(* CoDeSys 2.3.9.62 project: DosVagones.pro *)
(* Libraries: Standard.lib 2.6.14 10:37:46, IecSfc.lib 2.6.14 11:37:46 *)

(* Global variable list: Global_Variables *)
VAR_GLOBAL

      (*Entradas*)
      P1:BOOL;
      P2:BOOL;
	A1:BOOL;
	B1:BOOL;
	A2:BOOL;
	B2:BOOL;

       (* Salidas *)
	MOTOR_IZ1:BOOL;
	MOTOR_DE1:BOOL;
       MOTOR_IZ2:BOOL;
	MOTOR_DE2:BOOL;
      Carga1:BOOL;
      Carga2:BOOL;
      Descarga1:BOOL;
      Descarga2:BOOL;

      (* Variables del simulador *)
	Vel:INT:=1;
	Vel2:INT:=1;
END_VAR

(* POU PLC_PRG, ST *)
PROGRAM PLC_PRG
VAR
END_VAR
Vehiculo();
Vehiculo2();

Automatismo;
END_PROGRAM

(* POU Vehiculo, ST *)
PROGRAM Vehiculo
VAR
	PosX: INT;
END_VAR
A1:=FALSE;
B1:=FALSE;


IF MOTOR_DE1=TRUE THEN

     PosX:=PosX+Vel;

END_IF

IF MOTOR_IZ1=TRUE THEN

     PosX:=PosX-Vel;

END_IF


IF PosX<=0 THEN
   A1:=TRUE;
END_IF

IF PosX>=400 THEN
  B1:=TRUE;
END_IF
END_PROGRAM

(* POU Vehiculo2, ST *)
PROGRAM Vehiculo2
VAR
	PosX2: INT;
END_VAR
A2:=FALSE;
B2:=FALSE;


IF MOTOR_DE2=TRUE THEN

     PosX2:=PosX2+Vel2;

END_IF

IF MOTOR_IZ2=TRUE THEN

     PosX2:=PosX2-Vel2;

END_IF


IF PosX2<=0 THEN
   A2:=TRUE;
END_IF

IF PosX2>=400 THEN
  B2:=TRUE;
END_IF
END_PROGRAM

(* POU Automatismo, LD *)
PROGRAM Automatismo
VAR
	Control1: controlVehiculo;
	Control2: ControlVehiculo;
	IniciaDescarga: BOOL;
	EnB2: BOOL;
	EnB1: BOOL;
END_VAR
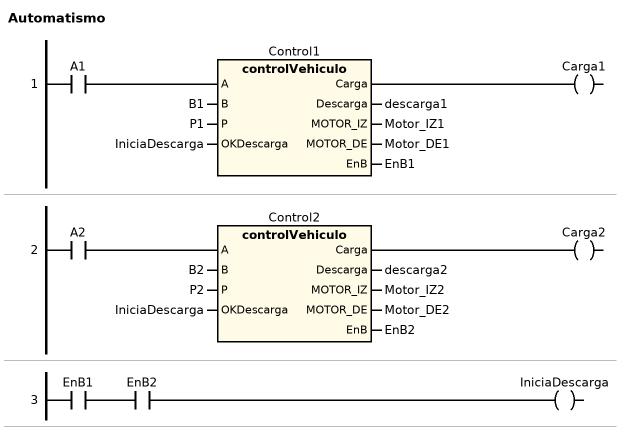
_LD_ (* Ladder Diagram *)
NETWORK 1
	[A1] - Control1:controlVehiculo(A: *, B: B1, P: P1, OKDescarga: IniciaDescarga, Descarga => descarga1, MOTOR_IZ => Motor_IZ1, MOTOR_DE => Motor_DE1, EnB => EnB1) --- (Carga1)
NETWORK 2
	[A2] - Control2:controlVehiculo(A: *, B: B2, P: P2, OKDescarga: IniciaDescarga, Descarga => descarga2, MOTOR_IZ => Motor_IZ2, MOTOR_DE => Motor_DE2, EnB => EnB2) --- (Carga2)
NETWORK 3
	[EnB1] - [EnB2] --- (IniciaDescarga)
_END_LD_
(* the same logic as Structured Text *)
(* Network 1 *)
Control1(A := A1, B := B1, P := P1, OKDescarga := IniciaDescarga);
descarga1 := Control1.Descarga;
Motor_IZ1 := Control1.MOTOR_IZ;
Motor_DE1 := Control1.MOTOR_DE;
EnB1 := Control1.EnB;
Carga1 := Control1.Carga;
(* Network 2 *)
Control2(A := A2, B := B2, P := P2, OKDescarga := IniciaDescarga);
descarga2 := Control2.Descarga;
Motor_IZ2 := Control2.MOTOR_IZ;
Motor_DE2 := Control2.MOTOR_DE;
EnB2 := Control2.EnB;
Carga2 := Control2.Carga;
(* Network 3 *)
IniciaDescarga := EnB1 AND EnB2;
END_PROGRAM

(* POU ControlVehiculo, LD *)
FUNCTION_BLOCK ControlVehiculo
VAR_INPUT
	A: BOOL;
	B: BOOL;
	P: BOOL;
	OKDescarga: BOOL;
END_VAR
VAR_OUTPUT
	Carga: BOOL;
	Descarga: BOOL;
	MOTOR_IZ: BOOL;
	MOTOR_DE: BOOL;
	EnB: BOOL;
END_VAR
VAR
	TCarga: TON;
	TDescarga: TON;
	T4s: BOOL;
END_VAR
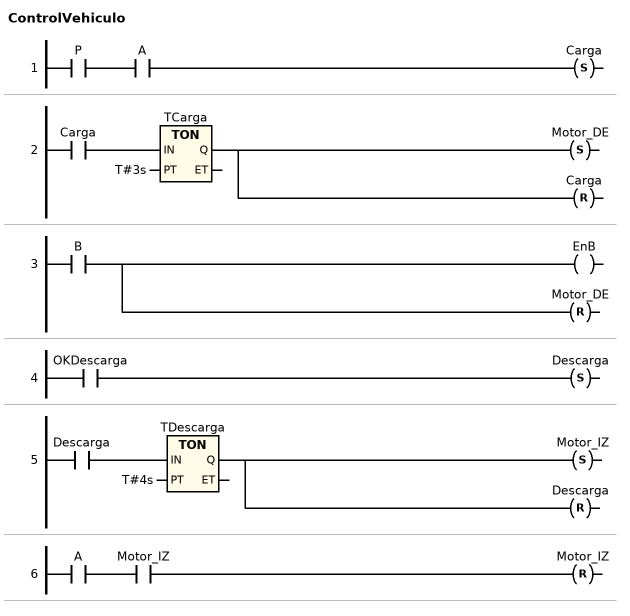
_LD_ (* Ladder Diagram *)
NETWORK 1
	[P] - [A] --- (S Carga)
NETWORK 2
	[Carga] - TCarga:TON(IN: *, PT: T#3s) --- (S Motor_DE) (R Carga)
NETWORK 3
	[B] --- (EnB) (R Motor_DE)
NETWORK 4
	[OKDescarga] --- (S Descarga)
NETWORK 5
	[Descarga] - TDescarga:TON(IN: *, PT: T#4s) --- (S Motor_IZ) (R Descarga)
NETWORK 6
	[A] - [Motor_IZ] --- (R Motor_IZ)
_END_LD_
(* the same logic as Structured Text *)
(* Network 1 *)
IF P AND A THEN Carga := TRUE; END_IF;
(* Network 2 *)
TCarga(IN := Carga, PT := T#3s);
IF TCarga.Q THEN Motor_DE := TRUE; Carga := FALSE; END_IF;
(* Network 3 *)
EnB := B;
IF B THEN Motor_DE := FALSE; END_IF;
(* Network 4 *)
IF OKDescarga THEN Descarga := TRUE; END_IF;
(* Network 5 *)
TDescarga(IN := Descarga, PT := T#4s);
IF TDescarga.Q THEN Motor_IZ := TRUE; Descarga := FALSE; END_IF;
(* Network 6 *)
IF A AND Motor_IZ THEN Motor_IZ := FALSE; END_IF;
END_FUNCTION_BLOCK

(* Visualisation Vehiculo
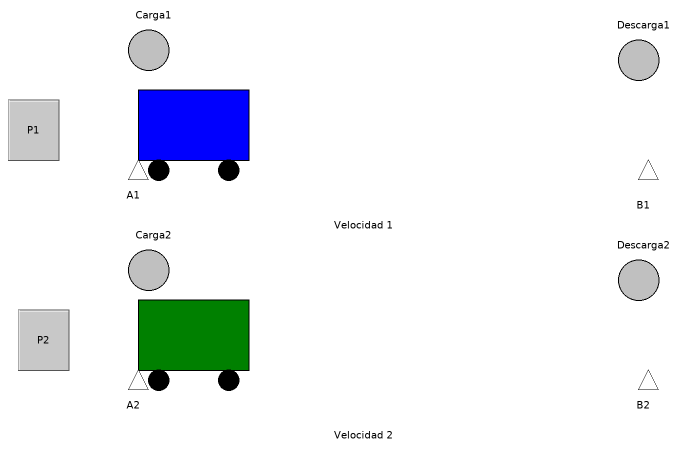
rectangle at (140,120)-(251,191): x offset Vehiculo.PosX
polygon at (130,190)-(150,210): alarm colour if .A1
polygon at (640,190)-(660,210): alarm colour if .B1
button at (10,130)-(61,191): text "P1"; taps P1
rectangle at (140,330)-(251,401): x offset Vehiculo2.PosX2
polygon at (130,400)-(150,420): alarm colour if .A2
polygon at (640,400)-(660,420): alarm colour if .B2
ellipse at (150,190)-(171,211): x offset Vehiculo.PosX
ellipse at (220,190)-(241,211): x offset Vehiculo.PosX
ellipse at (150,400)-(171,421): x offset Vehiculo2.PosX2
ellipse at (220,400)-(241,421): x offset Vehiculo2.PosX2
rectangle at (310,240)-(421,271): text "Velocidad 1"
rectangle at (310,450)-(421,481): text "Velocidad 2"
rectangle at (120,210)-(151,241): text "A1"
rectangle at (120,420)-(151,451): text "A2"
rectangle at (630,220)-(661,251): text "B1"
rectangle at (630,420)-(661,451): text "B2"
ellipse at (130,60)-(171,101): alarm colour if Carga1
rectangle at (100,30)-(211,61): text "Carga1"
ellipse at (130,280)-(171,321): alarm colour if Carga2
rectangle at (100,250)-(211,281): text "Carga2"
button at (20,340)-(71,401): text "P2"; taps P2
ellipse at (620,70)-(661,111): alarm colour if Descarga1
rectangle at (590,40)-(701,71): text "Descarga1"
ellipse at (620,290)-(661,331): alarm colour if Descarga2
rectangle at (590,260)-(701,291): text "Descarga2"
2 elements of other kinds (tables, trends, ...) not read
*)
